// Mitsubishi GX Works2 project: 02SignalLight   PLC: Q02U

PROGRAM MAIN
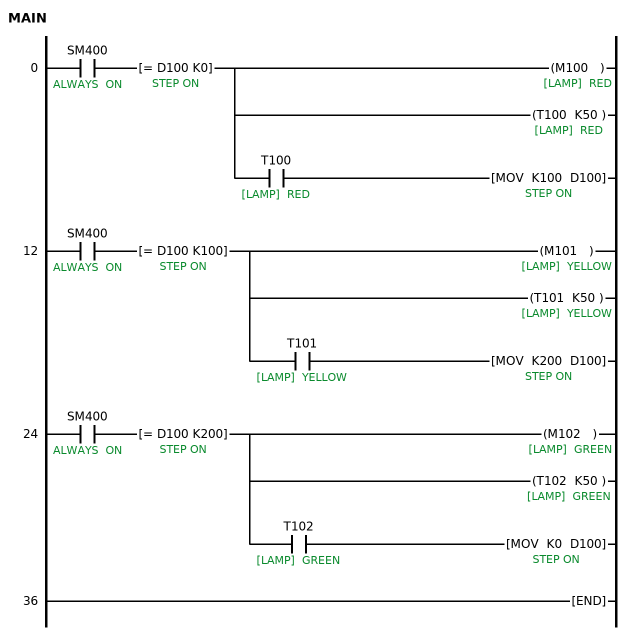
0     LD      SM400  ; ALWAYS  ON
      AND=    D100 K0  ; STEP ON
      OUT     M100  ; [LAMP]  RED
      OUT     T100 K50  ; [LAMP]  RED
      AND     T100  ; [LAMP]  RED
      MOV     K100 D100
12    LD      SM400  ; ALWAYS  ON
      AND=    D100 K100  ; STEP ON
      OUT     M101  ; [LAMP]  YELLOW
      OUT     T101 K50  ; [LAMP]  YELLOW
      AND     T101  ; [LAMP]  YELLOW
      MOV     K200 D100
24    LD      SM400  ; ALWAYS  ON
      AND=    D100 K200  ; STEP ON
      OUT     M102  ; [LAMP]  GREEN
      OUT     T102 K50  ; [LAMP]  GREEN
      AND     T102  ; [LAMP]  GREEN
      MOV     K0 D100
36    END
END_PROGRAM

PROGRAM LAMP
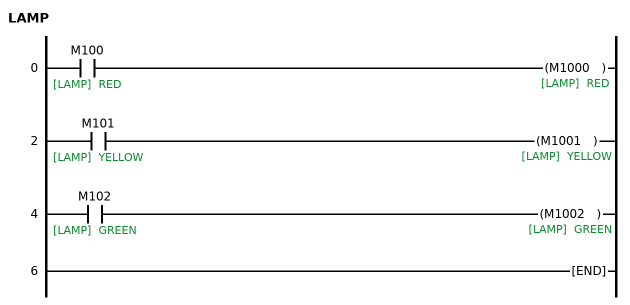
0     LD      M100  ; [LAMP]  RED
      OUT     M1000  ; [LAMP]  RED
2     LD      M101  ; [LAMP]  YELLOW
      OUT     M1001  ; [LAMP]  YELLOW
4     LD      M102  ; [LAMP]  GREEN
      OUT     M1002  ; [LAMP]  GREEN
6     END
END_PROGRAM

// device comments not shown above
M0  ; TIMER   TEST
T0  ; TIMER   TEST
